# EPICS alarm handler configuration: css_share/detectors/SVT/alh/SVT.R1.alhConfig
GROUP NULL R1
INCLUDE R1 SVT.R1.S1.alhConfig
INCLUDE R1 SVT.R1.S2.alhConfig
INCLUDE R1 SVT.R1.S3.alhConfig
INCLUDE R1 SVT.R1.S4.alhConfig
INCLUDE R1 SVT.R1.S5.alhConfig
INCLUDE R1 SVT.R1.S6.alhConfig
INCLUDE R1 SVT.R1.S7.alhConfig
INCLUDE R1 SVT.R1.S8.alhConfig
INCLUDE R1 SVT.R1.S9.alhConfig
INCLUDE R1 SVT.R1.S10.alhConfig
